// TIA Portal V20 export
DATA_BLOCK "DatafromFlinkToSafety"   // DB210
// stored: InstanceOfName Safety.typeDatafromFlinkToSafety, InstanceOfType UDT, Namespace Safety
"Safety.typeDatafromFlinkToSafety"
   // VAR
   //    "RcvBuffer.BA10" : Array[0..1, 0..121] of Byte;
   //    "ReceivedData.BA10" : Array[0..121] of Byte;
   //    "ReceivedAck.BA10" : Array[0..121] of Byte;
   //    "RcvBuffer.BA15" : Array[0..1, 0..121] of Byte;
   //    "ReceivedData.BA15" : Array[0..121] of Byte;
   //    "ReceivedAck.BA15" : Array[0..121] of Byte;
   //    "RcvBuffer.BA40" : Array[0..1, 0..121] of Byte;
   //    "ReceivedData.BA40" : Array[0..121] of Byte;
   //    "ReceivedAck.BA40" : Array[0..121] of Byte;
   //    "RcvBuffer.BA60" : Array[0..1, 0..121] of Byte;
   //    "ReceivedData.BA60" : Array[0..121] of Byte;
   //    "ReceivedAck.BA60" : Array[0..121] of Byte;
   // END_VAR
BEGIN
END_DATA_BLOCK
